(* CODESYS project myproject.project

Project tree, tasks and I/O mapping:
  CODESYS_Control_for_Raspberry_Pi : CODESYS Control for Raspberry Pi, 3S - Smart Software Solutions GmbH, version 3.5.10.0
    application Application
      libraries: Util, * (System)
      task MainTask (cyclic, interval t#10ms, priority 1) calls PLC_Logic
      program PLC_Logic [ST]
    SoftMotion General Axis Pool
    GPIOs_A_B : GPIOs A/B, 3S - Smart Software Solutions GmbH, version 1.1.1.10
        input  dIn : DWORD  // digital inputs (GPIO0..GPIO31)
        output dOut : DWORD  // digital outputs (GPIO0..GPIO31)
    Camera device
      <Empty>
    I²C
      I2C_master : I2C master, 3S - Smart Software Solutions GmbH, version 1.0.0.0
        Adafruit_PWM : Adafruit PWM, 3S - Smart Software Solutions GmbH, version 1.2.0.0
    SPI
    Onewire
  libraries: VisuSymbols, 3.5.10.0 (System)
  text list GlobalTextList
*)

// CODESYS_Control_for_Raspberry_Pi/Application/PLC_Logic
PROGRAM PLC_Logic
VAR CONSTANT
	PI: LREAL := 3.141592653589793;
END_VAR
VAR
	button: BOOL;
	led: BOOL;
	counter: INT := 0;
	t: LREAL := 0;
END_VAR

// Assuming a scan cycle of 10ms
// If button is not pressed (true)
//  - LED toggles every 2 seconds
//  - Servo completes a round (forward and backward) in 2 seconds
// If button is pressed (false), the frquency is multiplied by four, so:
//  - LED toggles every 500 milliseconds
//  - Servo completes a round in 500 milliseconds
button := dIn.24;
IF (button) THEN
	counter := counter + 1;
	t := t + PI * 2 / 200.0;
ELSE
	counter := counter + 4;
	t := t + PI * 2 / 50.0;
END_IF

// Controlling the Servo Motor With a Sinus Wave (Forward-Backward)
Adafruit_PWM.alrPWM[0] := 0.45 + 0.5 * SIN(t);

// Controlling LED and reset counters
IF (counter >= 200) THEN
	led := NOT led;
	dOut.22 := led;
	counter := 0;
	t := 0.0;
END_IF

END_PROGRAM
